// TIA Portal V20 export
TYPE "UDT_MTP_MonAnaDrv"
TITLE = MTPDataObjectSUCLibrary/DataAssembly/AnaDrv
   STRUCT
      FwdEn { ExternalWritable := 'False'} : Bool := FALSE;   // Forward movement enable1: enabled0: disabled
      RevEn { ExternalWritable := 'False'} : Bool := FALSE;   // Reverse movement enable1: enabled0: disabled
      StopOp : Bool := FALSE;   // Stop Command from Operator (relevant, if StateOpAct) 0-->1:request from POL 1-->0:acknowledge from PEA (Handshake)
      FwdOp : Bool := FALSE;   // Forward Command from Operator (relevant, if StateOpAct & FwdEn) 0-->1: request from POL 1-->0: acknowledge from PEA (Handshake)
      RevOp : Bool := FALSE;   // Reverse Command from Operator (relevant, if StateOpAct & RevEn) 0-->1: request from POL 1-->0: acknowledge from PEA (Handshake)
      OSLevel : Byte := 16#00;   // OSLevel variable
      StateChannel { ExternalWritable := 'False'} : Bool;   // Selection of the active OperationMode interaction channel0: The operator switches (*Op) shall be used.1: The automatic switches (*Aut) shall be used.
      StateOffAut { ExternalWritable := 'False'} : Bool;   // Set OperationMode to Offline by automatic interaction (relevant, if StateChannel).1: OperationMode is set to Offline.0: no operation
      StateOffOp : Bool;   // Set OperationMode to Offline by operator interaction (relevant, if not StateChannel) 0-->1:request to set OperationMode to Offline 1-->0:acknowledge by PEA
      StateOpAut { ExternalWritable := 'False'} : Bool;   // Set OperationMode to Operator by automatic interaction (relevant, if StateChannel).1: OperationMode is set to Manual.0: no operation
      StateOpOp : Bool;   // Set OperationMode to Operator by operator interaction (relevant, if not StateChannel) 0-->1:request to set OperationMode to Manual 1-->0:acknowledge by PEA
      StateAutAut { ExternalWritable := 'False'} : Bool;   // Set OperationMode to Automatic by automatic interaction (relevant, if StateChannel).1: OperationMode is set to Automatic.0: no operation
      StateAutOp : Bool;   // Set OperationMode to Automatic by operator interaction (relevant, if not StateChannel) 0-->1:request to set OperationMode is to Automatic 1-->0:acknowledge by PEA
      StateOpAct { ExternalWritable := 'False'} : Bool;   // 1: current mode is Operator0: current mode is not Operator
      StateAutAct { ExternalWritable := 'False'} : Bool;   // 1: current mode is Automatic0: current mode is not Automatic
      StateOffAct { ExternalWritable := 'False'} : Bool;   // 1: current mode is Offline0: current mode is not Offline
      SrcChannel { ExternalWritable := 'False'} : Bool;   // selection of the active SourceMode interaction channel0: The operator switches (*Op) shall be used.1: The automatic switches (*Aut) shall be used
      SrcManAut { ExternalWritable := 'False'} : Bool;   // Set SourceMode to Manual by automatic interaction (relevant, if SrcChannel).1: SourceMode is set to Manual.0: no operation
      SrcIntAut { ExternalWritable := 'False'} : Bool;   // Set SourceMode to Internal by automatic interaction (relevant, if SrcChannel).1: SourceMode is set to Internal.0: no operation
      SrcIntOp : Bool;   // Set SourceMode to Internal by operator interaction (relevant, if SrcChannel is false) 0-->1:request to set OperationMode to Internal 1-->0:acknowledge by PEA
      SrcManOp : Bool;   // Set SourceMode to Manual by operator interaction (relevant, if SrcChannel is false) 0-->1:request to set OperationMode to Manual 1-->0:acknowledge by PEA
      SrcIntAct { ExternalWritable := 'False'} : Bool;   // 1: current mode is Internal0: current mode is not Internal
      SrcManAct { ExternalWritable := 'False'} : Bool;   // 1: current mode is Manual0: current mode is not Manual
      SafePos { ExternalWritable := 'False'} : Bool := FALSE;   // Safe Position1: running0: stopped
      SafePosAct { ExternalWritable := 'False'} : Bool := FALSE;   // Safe Position activated 1: Safe Position is activated (safe operation) 0: Safe Position is not activated (normal operation)
      CSF { ExternalWritable := 'False'} : Bool;   // Reserved
      WQC { ExternalWritable := 'False'} : Byte := 16#FF;   // Worst Quality Code variable
      StopAut { ExternalWritable := 'False'} : Bool := FALSE;   // Set Drive to Stop by automatic.(relevant, if StateAutAct)1: Stop Command executed0: no operation
      FwdAut { ExternalWritable := 'False'} : Bool := FALSE;   // Set Drive to Forward by Automatic (relevant, if StateAutAct & FwdEn) 1:forward request 0:no forward request
      RevAut { ExternalWritable := 'False'} : Bool := FALSE;   // Set Drive to Reverse by Automatic (relevant, if StateAutAct & RevEn) 1:reverse request 0:no reverse request
      FwdCtrl { ExternalWritable := 'False'} : Bool := FALSE;   // Forward Control1: active0: inactive
      RevCtrl { ExternalWritable := 'False'} : Bool := FALSE;   // Reverse Control1: active0: inactive
      RevFbkCalc { ExternalWritable := 'False'} : Bool;   // Reverse Feedback Source1: calculated0: sensor detection
      FwdFbkCalc { ExternalWritable := 'False'} : Bool;   // Forward Feedback Source1: calculated0: sensor detection
      RpmFbkCalc { ExternalWritable := 'False'} : Bool;   // RPM Feedback Source1: calculated0: sensor detection
      RevFbk { ExternalWritable := 'False'} : Bool;   // Reverse Feedback Signal1: reverse running0: is not reverse running
      FwdFbk { ExternalWritable := 'False'} : Bool;   // Forward Feedback Signal1: forward running0: is not forward running
      Trip { ExternalWritable := 'False'} : Bool := FALSE;   // Drive Protection Indicator1: no problem0: Drive Protection triggered
      RpmSclMin { ExternalWritable := 'False'} : Real := 0.0;   // RPM Setpoint Scale Low Limit
      RpmSclMax { ExternalWritable := 'False'} : Real := 100.0;   // RPM Setpoint Scale High Limit
      RpmUnit { ExternalWritable := 'False'} : Int := 1001;   // RPM Setpoint Unit
      RpmMan : Real := 0.0;   // (relevant, if SrcManAct)RPM Manual Setpoint
      RpmInt { ExternalWritable := 'False'} : Real := 0.0;   // (relevant, if SrcIntAct)RPM Internal Setpoint
      RpmMin { ExternalWritable := 'False'} : Real := 0.0;   // RPM Setpoint Low Limit
      RpmMax { ExternalWritable := 'False'} : Real := 100.0;   // RPM Setpoint High Limit
      Rpm { ExternalWritable := 'False'} : Real := 0.0;   // RPM Setpoint
      RpmRbk { ExternalWritable := 'False'} : Real := 0.0;   // RPM Readback
      RpmFbk { ExternalWritable := 'False'} : Real := 0.0;   // RPM Feedback Signal
      PermEn { ExternalWritable := 'False'} : Bool := FALSE;   // Enables the Permission Lock1: enabled0: disabled
      Permit { ExternalWritable := 'False'} : Bool := FALSE;   // Permit allows control1: permission is given0: permission is not given
      IntlEn { ExternalWritable := 'False'} : Bool := FALSE;   // Enables the Interlock Lock1: enabled0: disabled
      Interlock { ExternalWritable := 'False'} : Bool := FALSE;   // Interlock prevents from being activated and sets it to safe position1: Interlock is not active0: Interlock is active
      ProtEn { ExternalWritable := 'False'} : Bool := FALSE;   // Enables the Protection Lock1: enabled; 0: disabled
      Protect { ExternalWritable := 'False'} : Bool := FALSE;   // Protect prevents from being activated and sets it to safe position, requires a reset command1: protect is not active0: protect is active, requires reset
      ResetOp : Bool := FALSE;   // Reset from Operator 0-->1:request from POL 1-->0:acknowledge from PEA (see Handshake)
      ResetAut { ExternalWritable := 'False'} : Bool := FALSE;   // Reset from Automatic 1:Reset execute 0:no operation
      MonEn : Bool := FALSE;   // Monitor Enable1: enabled0: disabled
      MonSafePos { ExternalWritable := 'False'} : Bool;   // Set the Error Behavior, if an error occurs.1: After an error occurs, the safe pos will be set.0: After an error occurs, the entity holds the state.
      MonStatErr { ExternalWritable := 'False'} : Bool := FALSE;   // Static Error active1: active0: inactive
      MonDynErr { ExternalWritable := 'False'} : Bool := FALSE;   // Dynamic Error active1: active0: inactive
      MonStatTi { ExternalWritable := 'False'} : Real := 0.0;   // Monitor Time for uncontrolled changes, in s
      MonDynTi { ExternalWritable := 'False'} : Real := 0.0;   // Monitor Time for controlled changes, in s
      RpmErr { ExternalWritable := 'False'} : Real := 0.0;   // RPM Error (RpmErr = Rpm – RpmFbk)
      RpmAHEn { ExternalWritable := 'False'} : Bool := FALSE;   // Enable Alarm High Limit1: enabled0: disabled
      RpmALEn { ExternalWritable := 'False'} : Bool := FALSE;   // Enable Alarm Low Limit1: enabled0: disabled
      RpmAHAct { ExternalWritable := 'False'} : Bool := FALSE;   // Alarm High Active 1:enabled 0:disabled
      RpmALAct { ExternalWritable := 'False'} : Bool := FALSE;   // Alarm Low Active 1:enabled 0:disabled
      RpmAHLim : Real := 100.0;   // Limit Value for Alarm High
      RpmALLim : Real := 0.0;   // Limit Value for Alarm Low
      StartingFbk { ExternalWritable := 'False'} : Bool := FALSE;   // Reserved
      StoppingFbk { ExternalWritable := 'False'} : Bool := FALSE;   // Reserved
   END_STRUCT;
END_TYPE
